{attribute 'pack_mode' := '1'}
TYPE ST_ReadListData_Array :
STRUCT
	stReadListReturnInfo	: ARRAY [1..2] OF ST_UAReadListReturnInfo;
	iArrayIntVar1 			: ARRAY[0..9] OF DINT;
	iArrayIntVar2 			: ARRAY[0..9] OF DINT;
END_STRUCT
END_TYPE

(* stored: Version 1.1.0.1
   DUT ST_ReadListData_Array: Id {1745a3a2-70fa-4aa5-9950-79e4b7b5d76e} *)
